Fanuc KAREL source: ka00134.KL

-- PROVISIONAL review KL for V770-1; original PC SHA256 96f81b33fc133957065fad75679bae938e27259629ccf7ab6375c98289d204bf
-- Incomplete behavior may be omitted. Consult companion uncertainty JSON. Do not deploy.
PROGRAM KA00134
%NOLOCKGROUP
VAR
  DST : REAL
-- UNRESOLVED_DECL SRC type=002017
BEGIN
  -- UNRESOLVED_PC offsets 5-19; opcodes 2E,22,9D,33,B4
  -- UNRESOLVED_PC offsets 24-40; opcodes 22,9D,33,B3,64,23
  -- UNRESOLVED_PC offsets 45-49; opcodes 7F
END KA00134
